Fanuc KAREL source: kd00054.KL

-- PROVISIONAL review KL for V770-1; original PC SHA256 3520ec961cbbd9472fd31b33e8aedcd1eb3c0691eb349aa703e6d0c422983ec1
-- Incomplete behavior may be omitted. Consult companion uncertainty JSON. Do not deploy.
PROGRAM KD00054
%NOLOCKGROUP
VAR
  I : INTEGER
  J : INTEGER
  B : BOOLEAN
  R : REAL
  S : STRING[80]
BEGIN
  -- UNRESOLVED_PC offsets 5-28; opcodes 9D,81,18,9D,1B,9D,12,22,2E,13,04
  -- UNRESOLVED_PC offsets 33-37; opcodes 7F
END KD00054
